FUNCTION_BLOCK FB_Motor
VAR_INPUT
END_VAR
VAR_OUTPUT
END_VAR
VAR
	
END_VAR

END_FUNCTION_BLOCK

(* stored: Version 1.1.0.1, ProductVersion 3.1.4024.16
   POU FB_Motor: Id {c81c8553-f5f9-451e-989a-9ec816095b07}, SpecialFunc None *)
